FUNCTION_BLOCK OR_6_BOOL (* FB to calculate boolean OR (generic FB) *)
  (* Standard: 61131-3; Classification: standard boolean function; Description: Copyright (c) 2014 Profactor GmbH This program and the accompanying materials are made available under the terms of the Eclipse Public License 2.0 which is available at https://www.eclipse.org/legal/epl-2.0/ SPDX-License-Identifier: EPL-2.0 *)
  (* Version 1.0, 2014-10-11, Matthias Plasch, Profactor GmbH *)
  (* Version 3.0, 2025-04-14, Patrick Aigner, changed package *)
  PACKAGE iec61131::bitwiseOperators;
  {SET_ATTRIBUTE(eclipse4diac::core::GenericClassName, 'GEN_OR')}
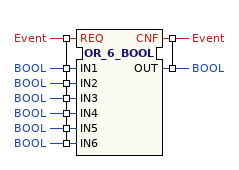
  EVENT_INPUT
    REQ WITH IN1, IN2, IN3, IN4, IN5, IN6; (* Normal Execution Request *)
  END_EVENT
  EVENT_OUTPUT
    CNF WITH OUT; (* Execution Confirmation *)
  END_EVENT
  VAR_INPUT
    IN1 : BOOL; (* OR input 1 *)
    IN2 : BOOL; (* OR input 2 *)
    IN3 : BOOL; (* OR input 3 *)
    IN4 : BOOL; (* OR input 4 *)
    IN5 : BOOL; (* OR input 5 *)
    IN6 : BOOL; (* OR input 6 *)
  END_VAR
  VAR_OUTPUT
    OUT : BOOL; (* OR result *)
  END_VAR
END_FUNCTION_BLOCK
